PROGRAM MAIN
VAR
	bRunOnlyOnce:BOOL:=FALSE;
	fOneFloat: REAL;
	sThisIsString: STRING;
	nAnInteger: INT;
	
	nReturnedNumberOfBytesForFloat: UDINT;
	nReturnedNumberOfBytesForString: UDINT;
	nReturnedNumberOfBytesForInteher: UDINT;
	stThisIsOurFirstUnstanceOfAStructure: ST_Event;
	bBoolean:BOOL:=FALSE;
END_VAR

IF NOT  bRunOnlyOnce THEN 
    ADSLOGDINT( msgCtrlMask := ADSLOG_MSGTYPE_ERROR OR ADSLOG_MSGTYPE_LOG, 
                    msgFmtStr := 'Hello, World!', dintArg:= 4711);
					bRunOnlyOnce:=TRUE;
END_IF	  
nReturnedNumberOfBytesForFloat:=SIZEOF(fOneFloat);
nReturnedNumberOfBytesForString:=SIZEOF(sThisIsString);
nReturnedNumberOfBytesForInteher:=SIZEOF(nAnInteger);

IF NOT bBoolean THEN
       UpdateEventTimestampWithSystemTime(stEvent:=stThisIsOurFirstUnstanceOfAStructure);
	   bBoolean:=TRUE;
END_IF;

END_PROGRAM

(* stored: Version 1.1.0.1, ProductVersion 3.1.4024.12
   POU MAIN: Id {f1417875-76a5-48aa-8ed5-dc97fff0b53e}, SpecialFunc None *)
